SUBAPPLICATION VT_active (* Subapplication Type *)
  (* Standard: 61499-2 *)
  (* Version 1.0, 2023-02-19, franz *)
  PACKAGE FBs::Counter::subs::page;
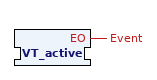
  EVENT_OUTPUT
    EO;
  END_EVENT
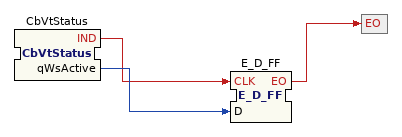
  FBS
    E_D_FF : iec61499::events::E_D_FF;
    CbVtStatus : isobus::UT::status::CbVtStatus;
  END_FBS
  EVENT_CONNECTIONS
    E_D_FF.EO TO EO;
    CbVtStatus.IND TO E_D_FF.CLK;
  END_CONNECTIONS
  DATA_CONNECTIONS
    CbVtStatus.qWsActive TO E_D_FF.D;
  END_CONNECTIONS
END_SUBAPPLICATION
